// Mitsubishi GX Works2 project: test_01   PLC: Q02/Q02H

// task Task_01 (event TRUE, interval 0, priority 31): POU_01

PROGRAM POU_01
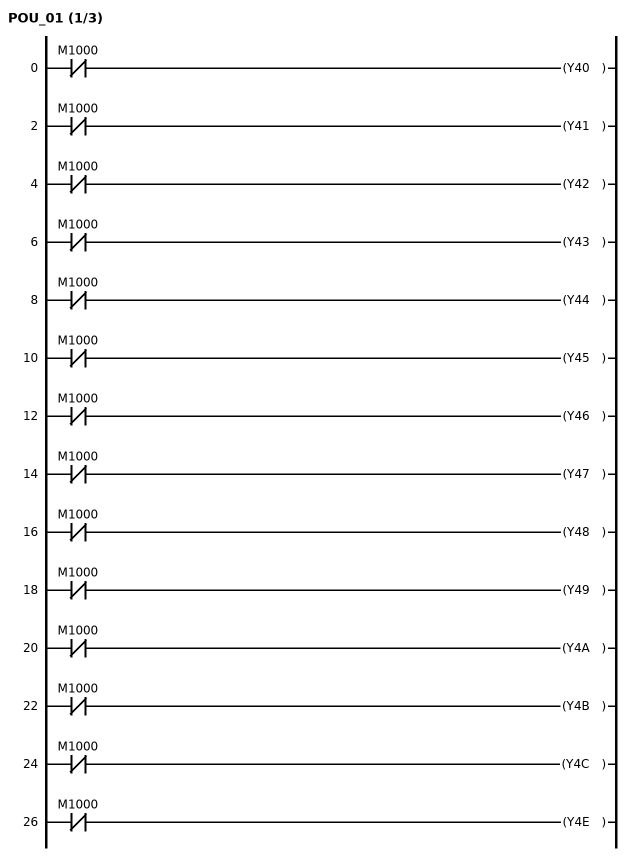
0     LDI     M1000
      OUT     Y40
2     LDI     M1000
      OUT     Y41
4     LDI     M1000
      OUT     Y42
6     LDI     M1000
      OUT     Y43
8     LDI     M1000
      OUT     Y44
10    LDI     M1000
      OUT     Y45
12    LDI     M1000
      OUT     Y46
14    LDI     M1000
      OUT     Y47
16    LDI     M1000
      OUT     Y48
18    LDI     M1000
      OUT     Y49
20    LDI     M1000
      OUT     Y4A
22    LDI     M1000
      OUT     Y4B
24    LDI     M1000
      OUT     Y4C
26    LDI     M1000
      OUT     Y4E
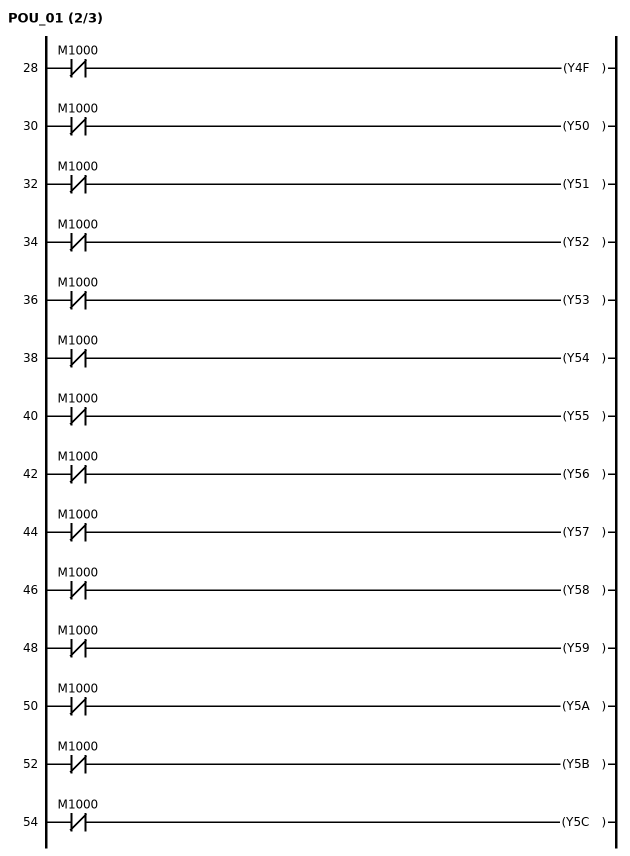
28    LDI     M1000
      OUT     Y4F
30    LDI     M1000
      OUT     Y50
32    LDI     M1000
      OUT     Y51
34    LDI     M1000
      OUT     Y52
36    LDI     M1000
      OUT     Y53
38    LDI     M1000
      OUT     Y54
40    LDI     M1000
      OUT     Y55
42    LDI     M1000
      OUT     Y56
44    LDI     M1000
      OUT     Y57
46    LDI     M1000
      OUT     Y58
48    LDI     M1000
      OUT     Y59
50    LDI     M1000
      OUT     Y5A
52    LDI     M1000
      OUT     Y5B
54    LDI     M1000
      OUT     Y5C
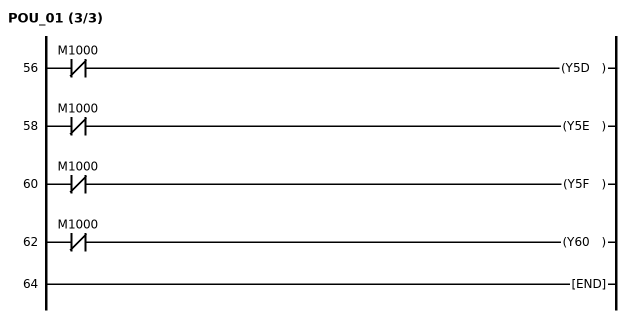
56    LDI     M1000
      OUT     Y5D
58    LDI     M1000
      OUT     Y5E
60    LDI     M1000
      OUT     Y5F
62    LDI     M1000
      OUT     Y60
64    END
END_PROGRAM
